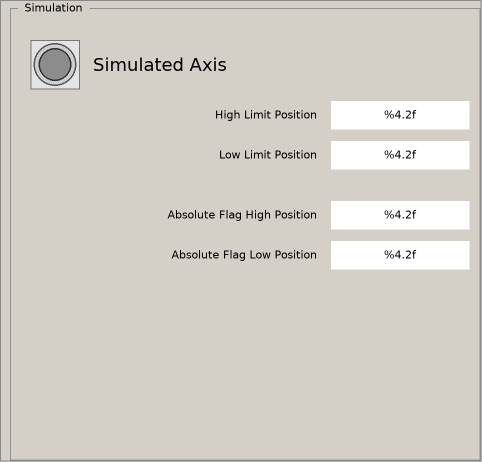
VISUALIZATION AxisSimulation  // 482x462
    GroupBox (10,0 470x460), "Simulation"
        PushSwitchLed (20,40 50x49), variable: MAIN.bSimulate[MAIN.hmiAxisSelect], behaviour: TOGGLE, style: Switch-PushSwitchLed-Gray
        Label (80,50 190x30), "Simulated Axis"
        Textfield (100,100 210x30), "High Limit Position", text variable: MAIN.hmiAxisSelect
        Textfield (320,100 140x30), "%4.2f", text variable: MAIN.simulated[MAIN.hmiAxisSelect].fHighLim
            OnMouseClick: write MAIN.simulated[MAIN.hmiAxisSelect].fHighLim via Default
        Textfield (100,140 210x30), "Low Limit Position", text variable: MAIN.hmiAxisSelect
        Textfield (320,240 140x30), "%4.2f", text variable: MAIN.simulated[MAIN.hmiAxisSelect].fLowAbs
            OnMouseClick: write MAIN.simulated[MAIN.hmiAxisSelect].fLowAbs via Default
    Textfield (330,140 140x30), "%4.2f", text variable: MAIN.simulated[MAIN.hmiAxisSelect].fLowLim
        OnMouseClick: write MAIN.simulated[MAIN.hmiAxisSelect].fLowLim via Default
    Textfield (110,200 210x30), "Absolute Flag High Position", text variable: MAIN.hmiAxisSelect
    Textfield (330,200 140x30), "%4.2f", text variable: MAIN.simulated[MAIN.hmiAxisSelect].fHighAbs
        OnMouseClick: write MAIN.simulated[MAIN.hmiAxisSelect].fHighAbs via Default
    Textfield (110,240 210x30), "Absolute Flag Low Position", text variable: MAIN.hmiAxisSelect
END_VISUALIZATION

(* stored: Version 1.1.0.1, ProductVersion 3.1.4022.12
   Visu AxisSimulation: Id {75e9ec67-a138-4c8a-ab6e-a53fc921a347} *)
